FUNCTION_BLOCK EL5021
VAR
	_io : EL5021_Data;
	{attribute addProperty Name "WcState"}
	_wcState : WcStateInputToggle;
	{attribute addProperty Name "Info data"}
	_infoData : InfoDataAdsDC;
END_VAR

PROPERTY IO : REFERENCE TO EL5021_Data
GET
IO REF= _io;
END_GET
END_PROPERTY

PROPERTY WcState : REFERENCE TO WcStateInputToggle
GET
WcState REF= _wcState;
END_GET
END_PROPERTY

END_FUNCTION_BLOCK

(* stored: Version 1.1.0.1, ProductVersion 3.1.4024.9
   POU EL5021: Id {345c6611-19ff-077f-3bfe-ba8ba76ade19}, SpecialFunc None
   Property IO: Id {76cd271f-13fe-0970-047b-9c7d5d7b19ea}
   Get Get: Id {7f256521-f27b-00be-1139-d564d8971fd4}
   Property WcState: Id {75c313a6-b4dc-0dcd-3637-9a5961c7b795}
   Get Get: Id {f2fe0719-60d2-06db-0370-120f170075ea} *)
